TYPE ST_ACDCCharger_events :
STRUCT
	b_CommunicationFault			:	BOOL;
	b_BuscouplerNotFound			:	BOOL;
	b_ACUnderVoltageDeratingActive	: 	BOOL;
	b_BatteryLimitDeratingActive	:	BOOL;
	b_TemperatureDeratingActive		:	BOOL;
	b_CurrentLimitActive			:	BOOL;
	b_SOCLimitReached				:	BOOL;
	b_FailedToGenerateDCOutput		:	BOOL;
	B_ACPhaselossFault				:	BOOL;
	B_ACUndervoltage				:	BOOL;
	B_ACOvervoltage					:	BOOL;
END_STRUCT
END_TYPE

(* stored: Version 1.1.0.1, ProductVersion 3.1.4026.18
   DUT ST_ACDCCharger_events: Id {3ea86631-6cb9-4920-a885-26748d7fabfd} *)
